Staubli VAL3: GetSNCtrl.pgx

program GetSNCtrl(string answer)
begin
//*******************************************************************************
//*   ______
//*  / _____) /|
//* | |      / /
//* | | /\  / /
//* | | \ \/ /  _      Copyright (c) KEOLABS, 2016
//* | |  \__/  | |        http://www.keolabs.com
//* | |________| |
//*  \__________/
//*
//********************************************************************************
//*@file          : GetSNCtrl
//*@author        : Yves Ragot
//*@version       : $Id: GetSNCtrl.pgx 1193 2016-10-06 09:55:11Z yves $
//*@brief         : Get Serial Number of the controller
//*
//*******************************************************************************/

  answer = left(getVersion("ControllerSN"), 20)

end
